Universal Robots PolyScope program: External_control.urp

Program External_control (installation=default directory=/programs createdIn=3.10.0.76181 lastSavedIn=3.10.0.76181 robotSerialNumber=2019351283)
Calibrated DH parameters: a=[0.000215, -0.418979, -0.391407, 0.000078, -0.000004, 0]; d=[0.089258, 26.735114, -28.945944, 2.320501, 0.094803, 0.082526]; alpha=[1.571788, 0.002752, 0.010358, 1.57059, -1.571136, 0]; deltaTheta=[0.000017, 0.173717, -0.232258, 0.058383, -0.000016, 0.000085]
Robot Program (runOnlyOnce=false)
  URCap External Control (External Control, FZI Research Center for Information Technology)
Event  expression=digital_out[0]≟ True
  Script: RG6(analog_out[0]*8750-35,analog_out[1]*6250)
  If tool_in[1]≟ True
    Set DigitalOutput pin=digital_out[0]; digitalValue=0
